// TIA Portal V19 export
TYPE "typeDevicesStatusSummary"
// General safety status of devices
// stored: Access Published, IsFailsafeCompliant true, Namespace Safety
   STRUCT
      allDevicesOk { ExternalWritable := 'False'} : Bool;   // All devices are released and acknowledged
      allEstopButtonsOK { ExternalWritable := 'False'} : Bool;   // All estop buttons are released and acknowledged
      allLighCurtainsOK { ExternalWritable := 'False'} : Bool;   // All light curtains are released and acknowledged
      allDoorsOK { ExternalWritable := 'False'} : Bool;   // All doors are released and acknowledged
      anyEstopButtonPressed { ExternalWritable := 'False'} : Bool;   // At least one estop button is pressed
      anyLightCurtainInterrupted { ExternalWritable := 'False'} : Bool;   // At least one light curtain is interrupted
      anyDoorOpen { ExternalWritable := 'False'} : Bool;   // At least one door is open
      anyDriveFault { ExternalWritable := 'False'} : Bool;   // At least one drive has a safety fault
      curtainsDisabled { ExternalWritable := 'False'} : Bool;   // Light curtains are disabled and inactive
      eStopDelayedOK { ExternalWritable := 'False'} : Bool;   // The delay estop OK signal is TRUE
   END_STRUCT;
END_TYPE
